FUNCTION_BLOCK E_UCNTR (* Basic Function Block Type *)
  (* Standard: 61499-2 *)
  (* Version 0.0, 2/8/2023, brink, Flexbridge AB, Template *)
  PACKAGE UAO.Hackathon;
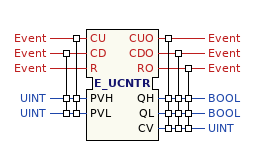
  EVENT_INPUT
    CU WITH PVH, PVL; (* Count up *)
    CD WITH PVH, PVL; (* Count down *)
    R;
  END_EVENT
  EVENT_OUTPUT
    CUO WITH QH, QL, CV; (* Execution Confirmation *)
    CDO WITH QH, QL, CV;
    RO WITH QH, QL, CV;
  END_EVENT
  VAR_INPUT
    PVH : UINT; (* Preset value high *)
    PVL : UINT; (* Preset value low *)
  END_VAR
  VAR_OUTPUT
    QH : BOOL; (* Output event qualifier *)
    QL : BOOL; (* Output event qualifier *)
    CV : UINT;
  END_VAR
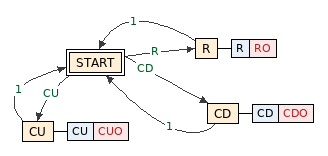
  EC_STATES
    START; (* Initial State *)
    CD : CD -> CDO; (* Normal execution *)
    CU : CU -> CUO;
    R : R -> RO;
  END_STATES
  EC_TRANSITIONS
    START TO CD := CD;
    START TO CU := CU;
    START TO R := R;
    R TO START := 1;
    CU TO START := 1;
    CD TO START := 1;
  END_TRANSITIONS
  ALGORITHM CU IN ST: (* Initialization algorithm *)
CV := CV + 1;
QL := CV <= PVL;
QH := CV >= PVH;
  END_ALGORITHM
  ALGORITHM CD IN ST: (* Normally executed algorithm *)
IF CV > 0 THEN
	CV := CV - 1;
	QL := CV <= PVL;
	QH := CV >= PVH;
END_IF;
  END_ALGORITHM
  ALGORITHM R IN ST:
CV := 0;
QL := FALSE;
QH := FALSE;
  END_ALGORITHM
  ALGORITHM CNT IN ST:
QL := CV <= PVL;
QH := CV >= PVH;
  END_ALGORITHM
END_FUNCTION_BLOCK
